TYPE stackerUnLoadSettings :
STRUCT PERSISTENT
	
	axisLength                :   REAL   := 625.0; 		    // макс ход на оста на стакера за модел HEX 24
	axisWorkSpeed             :	  REAL   := 200.0; 	        // скорост 
	axisInitSpeed			  :   REAL   := 200.0; 	        // скорост при движение нагоре (при init)
	axisAcc					  :   REAL   := 200.0 ;         // ускр.
	pallet                    :   ARRAY[1..Consts.MAX_RECIPE] OF palletParamsU; 

END_STRUCT
END_TYPE

(* stored: Version 1.1.0.1, ProductVersion 3.1.4024.3
   DUT stackerUnLoadSettings: Id {e85d8732-ab02-4de7-ab2b-f34358de4d7d} *)
